// Mitsubishi GX Works2 project: 8   PLC: FX2N/FX2NC

PROGRAM MAIN
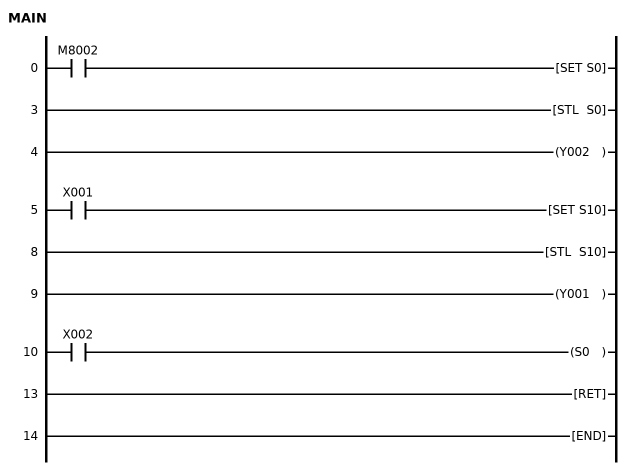
0     LD      M8002
      SET     S0
3     STL     S0
4     OUT     Y002
5     LD      X001
      SET     S10
8     STL     S10
9     OUT     Y001
10    LD      X002
      OUT     S0
13    RET
14    END
END_PROGRAM

// device comments not shown above
BL0  ; main
BL1  ; a
